{attribute 'qualified_only'}
{attribute 'strict'}
TYPE PunchingMachine :
(
	upward := 0,
	downward,
	switchoff
);
END_TYPE

(* stored: Version 1.1.0.1, ProductVersion 3.1.4022.12
   DUT PunchingMachine: Id {ed898153-0f71-4399-bcdc-50ff9a6deeb3} *)
